FUNCTION_BLOCK FB_SlitPairV2
VAR_INPUT
    nIdPositiveAxis: UINT; //ID of axis for which positive motion increases gap size
    nIdNegativeAxis: UINT; //ID of axis for which negative motion increases gap size
    nIdGapSizeAxis: UINT; //ID of virtual gap aperture size axis
    nIdGapCentreAxis: UINT; //ID of virtual gap centre position axis

    bEnable: BOOL; //Enable slit pair logic functionality
    bReset: BOOL; //Reset from error state
    fEncoderScaling: LREAL := 10000; //Virtual axis scaling denominator, default of 10000
END_VAR
VAR
    nGapSizeEncoder AT %Q*: UDINT := 0;
    nGapCentreEncoder AT %Q*: UDINT := 0;
    fGapSize: LREAL;
    fGapCentre: LREAL;
    bAllHalted: BOOL := FALSE;
    bInternalResetHome: BOOL :=FALSE;

    fbSetpointGenEnablePositiveAxis: MC_ExtSetPointGenEnable;
    fbSetpointGenEnableNegativeAxis: MC_ExtSetPointGenEnable;
    fbSetpointGenEnableGapSizeAxis: MC_ExtSetPointGenEnable;
    fbSetpointGenEnableGapCentreAxis: MC_ExtSetPointGenEnable;

    fbSetpointGenDisablePositiveAxis: MC_ExtSetPointGenDisable;
    fbSetpointGenDisableNegativeAxis: MC_ExtSetPointGenDisable;
    fbSetpointGenDisableGapSizeAxis: MC_ExtSetPointGenDisable;
    fbSetpointGenDisableGapCentreAxis: MC_ExtSetPointGenDisable;

    fPosSetpointPositiveAxis: LREAL;
    fPosSetpointNegativeAxis: LREAL;
    fPosSetpointGapSizeAxis: LREAL;
    fPosSetpointGapCentreAxis: LREAL;
    
    fPosSetpointPositiveAxis_Last: LREAL;
    fPosSetpointNegativeAxis_Last: LREAL;
    fPosSetpointGapSizeAxis_Last: LREAL;
    fPosSetpointGapCentreAxis_Last: LREAL;
    
    fPosSetpointPositiveAxis_Nominal: LREAL;
    fPosSetpointNegativeAxis_Nominal: LREAL;
    fPosSetpointGapSizeAxis_Nominal: LREAL;
    fPosSetpointGapCentreAxis_Nominal: LREAL;
    
    fPosSetpointPositiveAxis_New: LREAL;
    fPosSetpointNegativeAxis_New: LREAL;
    fPosSetpointGapSizeAxis_New: LREAL;
    fPosSetpointGapCentreAxis_New: LREAL;

    fVeloSetpointPositiveAxis: LREAL;
    fVeloSetpointNegativeAxis: LREAL;
    fVeloSetpointGapSizeAxis: LREAL;
    fVeloSetpointGapCentreAxis: LREAL;

    fVeloSetpointPositiveAxis_New: LREAL;
    fVeloSetpointNegativeAxis_New: LREAL;
    fVeloSetpointGapSizeAxis_New: LREAL;
    fVeloSetpointGapCentreAxis_New: LREAL;
    
    nDirectionPositiveAxis: DINT;
    nDirectionNegativeAxis: DINT;
    nDirectionGapSizeAxis: DINT;
    nDirectionGapCentreAxis: DINT;
    
    ePositiveAxisState : E_AxisLimitState;
    eNegativeAxisState : E_AxisLimitState;
    eAxisPairState : E_SlitPairLimitState;
    eSlitDirectionState : E_SlitDirectionState;
    

    eState: E_SlitPairStatesV2 := E_SlitPairStatesV2.eInit;

    bInternalReset: BOOL;
    bHomingReset: BOOL := FALSE;

    //Two resets required due to homing functionality
    bResetInProgressCheck1: BOOL := FALSE;
    bResetInProgressCheck2: BOOL := FALSE;

    //internal MCPOWER blocks because Beckhoff won't let you enable a setpoint generator on a limit....
    fbPowerPositiveAxis: MC_POWER;
    fbPowerNegativeAxis: MC_POWER;
    fbPowerGapSizeAxis: MC_POWER;
    fbPowerGapCentreAxis: MC_POWER;

    //internal MC_Reset, needed because the current reset in FB_Axis works only when there is an error. This should change once the reset functionality changes
    fbInternalResetTrig: R_TRIG;
    fbInternalResetHome: R_TRIG;
    fbResetPositiveAxis: MC_RESET;
    fbResetNegativeAxis: MC_RESET;
    fbResetGapSizeAxis: MC_RESET;
    fbResetGapCentreAxis: MC_RESET;
    fbResetHomedGap: MC_Home;
    fbResetHomedCentre: MC_Home;

END_VAR

(*SETUP INSTRUCTIONS
Virtual axes:
Encoder type set to Universal
Encoder mask set to 0xFFFFFFFF
Encoder scaling set to match FB
Link nDataIn1 of encoder to FB encoders
Position lag monitoring can be left on*
Dynamics of virtual axes must be configured considering coupled mechanicals (e.g. don't set velocities your real axes can't achieve)
Virtual axis limits will need to be much more state based, for example:
GAP SIZE fwd will only be disabled if +Ve fwd hit AND -ve bwd hit, not OR
*)

//Position of virtual axes
actVirtualAxisPositions();
//Limit logic
actLimitState();
actVirtualAxisLimits();

//*NOTES*/
(*
Might need to decouple virtual axis logic (i.e. let gap size increase even if centre position locked)
Will involve untracked movements, will involve NOT enabling certain setpoint generators in certain conditions or even 
disabling and enabling other generators during moves where necessary
i.e. a limit is hit trying to full open the gap size so disabled the centre setpoint generator and "gear it in" to the real axes


*)

//Enable Logic - Virtual axes automatically enable when real axes are enabled
actVirtualAxisEnable();
//Call spGenerator FBs
actGeneratorEnableDisable();
//Calculate position setpoints
actCalculateSetpointPositions();
//Calculate velocity setpoints
//actCalculateSetpointVelocities();
//Calculate directions
actCalculateSetpointDirections();

//Error state handling - only handle errors that disable motion
IF bEnable AND (GVL.astAxes[nIdPositiveAxis].Axis.Status.ErrorStop OR GVL.astAxes[nIdNegativeAxis].Axis.Status.ErrorStop OR GVL.astAxes[nIdGapSizeAxis].Axis.Status.ErrorStop OR GVL.astAxes[nIdGapCentreAxis].Axis.Status.ErrorStop) THEN
    //eState := E_SlitPairStatesV2.eError;
END_IF

//Propagate real axis error to virtual
IF GVL.astAxes[nIdPositiveAxis].Axis.Status.ErrorStop AND (NOT GVL.astAxes[nIdGapSizeAxis].Axis.Status.ErrorStop OR NOT GVL.astAxes[nIdGapCentreAxis].Axis.Status.ErrorStop) THEN
    //GVL.astAxes[nIdGapSizeAxis].stStatus.bError := TRUE;
    //GVL.astAxes[nIdGapCentreAxis].stStatus.bError := TRUE;
    GVL.astAxes[nIdGapSizeAxis].stStatus.nErrorID := GVL.astAxes[nIdPositiveAxis].stStatus.nErrorID;
    GVL.astAxes[nIdGapCentreAxis].stStatus.nErrorID := GVL.astAxes[nIdPositiveAxis].stStatus.nErrorID;
ELSIF  GVL.astAxes[nIdNegativeAxis].Axis.Status.ErrorStop AND (NOT GVL.astAxes[nIdGapSizeAxis].Axis.Status.ErrorStop OR NOT GVL.astAxes[nIdGapCentreAxis].Axis.Status.ErrorStop) THEN
    //GVL.astAxes[nIdGapSizeAxis].stStatus.bError := TRUE;
    //GVL.astAxes[nIdGapCentreAxis].stStatus.bError := TRUE;
    GVL.astAxes[nIdGapSizeAxis].stStatus.nErrorID := GVL.astAxes[nIdNegativeAxis].stStatus.nErrorID;
    GVL.astAxes[nIdGapCentreAxis].stStatus.nErrorID := GVL.astAxes[nIdNegativeAxis].stStatus.nErrorID;
END_IF

//Internal Reset linked to any axis reset
bInternalReset := bReset OR GVL.astAxes[nIdPositiveAxis].stControl.bReset OR GVL.astAxes[nIdNegativeAxis].stControl.bReset OR GVL.astAxes[nIdGapSizeAxis].stControl.bReset OR GVL.astAxes[nIdGapCentreAxis].stControl.bReset;

//If real axis is homing, change state
IF bEnable AND (GVL.astAxes[nIdPositiveAxis].Axis.Status.HomingBusy OR GVL.astAxes[nIdNegativeAxis].Axis.Status.HomingBusy) THEN
    eState := E_SlitPairStatesV2.eWaitForRealHomed;
END_IF

//Link all halt buttons in motors
IF GVL.astAxes[nIdPositiveAxis].stControl.bHalt OR GVL.astAxes[nIdNegativeAxis].stControl.bHalt OR
    GVL.astAxes[nIdGapSizeAxis].stControl.bHalt OR GVL.astAxes[nIdGapCentreAxis].stControl.bHalt THEN
    actHaltAllAxes();
END_IF

//Propagate homing status
fbResetHomedGap(Axis:= GVL.astAxes[nIdGapSizeAxis].Axis, HomingMode:= MC_ResetCalibration);
fbResetHomedCentre(Axis:= GVL.astAxes[nIdGapCentreAxis].Axis, HomingMode:= MC_ResetCalibration);
fbInternalResetHome(CLK:= fbResetHomedCentre.Done OR fbResetHomedGap.Done );
IF NOT GVL.astAxes[nIdPositiveAxis].stStatus.bHomed OR NOT GVL.astAxes[nIdNegativeAxis].stStatus.bHomed THEN
        fbResetHomedGap.Execute := TRUE;
        fbResetHomedCentre.Execute := TRUE;
END_IF

IF fbInternalResetHome.Q THEN
        fbResetHomedGap.Execute := FALSE;
        fbResetHomedCentre.Execute := FALSE;
END_IF


//State machine
IF bEnable THEN
    CASE eState OF  //HOMING LOOP ISSUE
        E_SlitPairStatesV2.eInit:
            //If real axes are calibrated, then home the virtual axes, else go Operatioanl
            fbResetPositiveAxis(Axis:=GVL.astAxes[nIdPositiveAxis].Axis, Execute:=FALSE);
            fbResetNegativeAxis(Axis:=GVL.astAxes[nIdNegativeAxis].Axis, Execute:=FALSE);
            fbResetGapSizeAxis(Axis:=GVL.astAxes[nIdGapSizeAxis].Axis, Execute:=FALSE);
            fbResetGapCentreAxis(Axis:=GVL.astAxes[nIdGapCentreAxis].Axis, Execute:=FALSE);
            IF GVL.astAxes[nIdPositiveAxis].stStatus.bHomed AND GVL.astAxes[nIdNegativeAxis].stStatus.bHomed THEN
               GVL.astAxes[nIdGapSizeAxis].stConfig.eHomeSeq := E_HomingRoutines.eHomeDirect;
               GVL.astAxes[nIdGapCentreAxis].stConfig.eHomeSeq := E_HomingRoutines.eHomeDirect;
               GVL.astAxes[nIdGapSizeAxis].stConfig.fHomePosition := fGapSize;
               GVL.astAxes[nIdGapCentreAxis].stConfig.fHomePosition := fGapCentre;
                eState := E_SlitPairStatesV2.eWaitForVirtualHomed;
            ELSE
                eState := E_SlitPairStatesV2.eOperational;
            END_IF

        E_SlitPairStatesV2.eWaitForVirtualHomed:
            //Wait for virtual axis homing to complete/
            GVL.astAxes[nIdGapSizeAxis].stControl.eCommand := E_MotionFunctions.eHome;
            GVL.astAxes[nIdGapSizeAxis].stControl.bExecute := TRUE;
            GVL.astAxes[nIdGapCentreAxis].stControl.eCommand := E_MotionFunctions.eHome;
            GVL.astAxes[nIdGapCentreAxis].stControl.bExecute := TRUE;
            IF GVL.astAxes[nIdGapSizeAxis].stStatus.bHomed AND GVL.astAxes[nIdGapCentreAxis].stStatus.bHomed THEN
                eState := E_SlitPairStatesV2.eOperational;
            END_IF
            //IF NOT IN HOMING STATE

        E_SlitPairStatesV2.eOperational:
            bResetInProgressCheck1 := FALSE;
            //Detect whether real or virtual axes are moving
            IF GVL.astAxes[nIdGapSizeAxis].stStatus.bMoving OR GVL.astAxes[nIdGapCentreAxis].stStatus.bMoving THEN
                eState := E_SlitPairStatesV2.eEnableRealGenerators;
            END_IF
            IF GVL.astAxes[nIdPositiveAxis].stStatus.bMoving OR GVL.astAxes[nIdNegativeAxis].stStatus.bMoving THEN
                eState := E_SlitPairStatesV2.eEnableVirtualGenerators;
            END_IF

        E_SlitPairStatesV2.eEnableRealGenerators:
            //Hold MC_Power on until generators have enabled
            fbPowerPositiveAxis(Axis:=GVL.astAxes[nIdPositiveAxis].Axis, Enable:=TRUE, Enable_Positive:=TRUE,Enable_Negative:=TRUE);
            fbPowerNegativeAxis(Axis:=GVL.astAxes[nIdNegativeAxis].Axis, Enable:=TRUE, Enable_Positive:=TRUE,Enable_Negative:=TRUE);
            fbSetpointGenEnablePositiveAxis.Execute := TRUE;
            fbSetpointGenEnableNegativeAxis.Execute := TRUE;
            eState := E_SlitPairStatesV2.eCheckRealAxisGeneratorsEnabled;

        E_SlitPairStatesV2.eCheckRealAxisGeneratorsEnabled:
            //Hold MC_Power on until generators have enabled
            fbPowerPositiveAxis(Axis:=GVL.astAxes[nIdPositiveAxis].Axis, Enable:=TRUE, Enable_Positive:=TRUE,Enable_Negative:=TRUE);
            fbPowerNegativeAxis(Axis:=GVL.astAxes[nIdNegativeAxis].Axis, Enable:=TRUE, Enable_Positive:=TRUE,Enable_Negative:=TRUE);
            IF fbSetpointGenEnablePositiveAxis.Enabled AND fbSetpointGenEnableNegativeAxis.Enabled THEN
                eState := E_SlitPairStatesV2.eWaitForVirtualMoveDone;
            END_IF

        E_SlitPairStatesV2.eWaitForVirtualMoveDone:            
            IF NOT(GVL.astAxes[nIdGapSizeAxis].stStatus.bMoving OR GVL.astAxes[nIdGapCentreAxis].stStatus.bMoving) THEN
                eState := E_SlitPairStatesV2.eDisableRealGenerators;
            END_IF

        E_SlitPairStatesV2.eDisableRealGenerators:
            fbSetpointGenDisablePositiveAxis.Execute := TRUE;
            fbSetpointGenDisableNegativeAxis.Execute := TRUE;
            eState := E_SlitPairStatesV2.eOperational;

        E_SlitPairStatesV2.eEnableVirtualGenerators:
            //Hold MC_Power on until generators have enabled
            fbPowerGapSizeAxis(Axis:=GVL.astAxes[nIdGapSizeAxis].Axis, Enable:=TRUE, Enable_Positive:=TRUE,Enable_Negative:=TRUE);
            fbPowerGapCentreAxis(Axis:=GVL.astAxes[nIdGapCentreAxis].Axis, Enable:=TRUE, Enable_Positive:=TRUE,Enable_Negative:=TRUE);
            fbSetpointGenEnableGapSizeAxis.Execute := TRUE;
            fbSetpointGenEnableGapCentreAxis.Execute := TRUE;
            eState := E_SlitPairStatesV2.eCheckVirtualAxisGeneratorsEnabled;

        E_SlitPairStatesV2.eCheckVirtualAxisGeneratorsEnabled:
            //Hold MC_Power on until generators have enabled
            fbPowerGapSizeAxis(Axis:=GVL.astAxes[nIdGapSizeAxis].Axis, Enable:=TRUE, Enable_Positive:=TRUE,Enable_Negative:=TRUE);
            fbPowerGapCentreAxis(Axis:=GVL.astAxes[nIdGapCentreAxis].Axis, Enable:=TRUE, Enable_Positive:=TRUE,Enable_Negative:=TRUE);
            IF fbSetpointGenEnableGapSizeAxis.Enabled AND fbSetpointGenEnableGapCentreAxis.Enabled THEN
                eState := E_SlitPairStatesV2.eWaitForRealMoveDone;
            END_IF

        E_SlitPairStatesV2.eWaitForRealMoveDone:
            IF NOT(GVL.astAxes[nIdPositiveAxis].stStatus.bMoving OR GVL.astAxes[nIdNegativeAxis].stStatus.bMoving) THEN
                eState := E_SlitPairStatesV2.eDisableVirtualGenerators;
            END_IF

        E_SlitPairStatesV2.eDisableVirtualGenerators:
            fbSetpointGenDisableGapSizeAxis.Execute := TRUE;
            fbSetpointGenDisableGapCentreAxis.Execute := TRUE;
            eState := E_SlitPairStatesV2.eOperational;

        E_SlitPairStatesV2.eError:
            actHaltAllAxes();

            IF bHomingReset THEN
                bInternalReset := TRUE;
                bResetInProgressCheck1 := TRUE;
                bResetInProgressCheck2 := TRUE;
                bHomingReset := FALSE;
            END_IF
            IF bInternalReset OR bReset OR bResetInProgressCheck2 THEN
                fbResetPositiveAxis(Axis:=GVL.astAxes[nIdPositiveAxis].Axis, Execute:=TRUE);
                fbResetNegativeAxis(Axis:=GVL.astAxes[nIdNegativeAxis].Axis, Execute:=TRUE);
                fbResetGapSizeAxis(Axis:=GVL.astAxes[nIdGapSizeAxis].Axis, Execute:=TRUE);
                fbResetGapCentreAxis(Axis:=GVL.astAxes[nIdGapCentreAxis].Axis, Execute:=TRUE);
                GVL.astAxes[nIdPositiveAxis].stControl.bReset := TRUE;
                GVL.astAxes[nIdNegativeAxis].stControl.bReset := TRUE;
                GVL.astAxes[nIdGapSizeAxis].stControl.bReset := TRUE;
                GVL.astAxes[nIdGapCentreAxis].stControl.bReset := TRUE;
                IF NOT(bResetInProgressCheck1) THEN
                    bResetInProgressCheck2 := FALSE;
                END_IF
            END_IF

            IF NOT(GVL.astAxes[nIdPositiveAxis].stStatus.bError) AND NOT(GVL.astAxes[nIdNegativeAxis].stStatus.bError) AND NOT(GVL.astAxes[nIdGapSizeAxis].stStatus.bError) AND NOT(GVL.astAxes[nIdGapCentreAxis].stStatus.bError) THEN
                eState := E_SlitPairStatesV2.eInit;
            END_IF

        E_SlitPairStatesV2.eWaitForRealHomed:
            bHomingReset := TRUE;
            IF NOT GVL.astAxes[nIdPositiveAxis].Axis.Status.Homed OR NOT GVL.astAxes[nIdNegativeAxis].Axis.Status.Homed THEN
                eState := E_SlitPairStatesV2.eInit;
            END_IF
    END_CASE
END_IF


//Feed externalsetpoint generators setpoint values - ignoring acceleration
MC_ExtSetPointGenFeed(Axis:= GVL.astAxes[nIdPositiveAxis].Axis, Position:= fPosSetpointPositiveAxis, Velocity:= fVeloSetpointPositiveAxis, Acceleration:= 0, Direction:= nDirectionPositiveAxis);
MC_ExtSetPointGenFeed(Axis:= GVL.astAxes[nIdNegativeAxis].Axis, Position:= fPosSetpointNegativeAxis, Velocity:= fVeloSetpointNegativeAxis, Acceleration:= 0, Direction:= nDirectionNegativeAxis);
MC_ExtSetPointGenFeed(Axis:= GVL.astAxes[nIdGapSizeAxis].Axis, Position:= fPosSetpointGapSizeAxis, Velocity:= fVeloSetpointGapSizeAxis, Acceleration:= 0, Direction:= nDirectionGapSizeAxis);
MC_ExtSetPointGenFeed(Axis:= GVL.astAxes[nIdGapCentreAxis].Axis, Position:= fPosSetpointGapCentreAxis, Velocity:= fVeloSetpointGapCentreAxis, Acceleration:= 0, Direction:= nDirectionGapCentreAxis);

bReset := FALSE;

ACTION actCalculateSetpointDirections:

IF fVeloSetpointPositiveAxis > 0 THEN
    nDirectionPositiveAxis := 1; //moving forward
ELSIF fVeloSetpointPositiveAxis < 0 THEN
    nDirectionPositiveAxis := -1; //moving backward
ELSE
    nDirectionPositiveAxis := 0; //stationary
END_IF

IF fVeloSetpointNegativeAxis > 0 THEN
    nDirectionNegativeAxis := 1; //moving forward
ELSIF fVeloSetpointNegativeAxis < 0 THEN
    nDirectionNegativeAxis := -1; //moving backward
ELSE
    nDirectionNegativeAxis := 0; //stationary
END_IF

IF fVeloSetpointGapSizeAxis > 0 THEN
    nDirectionGapSizeAxis := 1; //moving forward
ELSIF fVeloSetpointGapSizeAxis < 0 THEN
    nDirectionGapSizeAxis := -1; //moving backward
ELSE
    nDirectionGapSizeAxis := 0; //stationary
END_IF

IF fVeloSetpointGapCentreAxis > 0 THEN
    nDirectionGapCentreAxis := 1; //moving forward
ELSIF fVeloSetpointGapCentreAxis < 0 THEN
    nDirectionGapCentreAxis := -1; //moving backward
ELSE
    nDirectionGapCentreAxis := 0; //stationary
END_IF
END_ACTION

ACTION actCalculateSetpointPositions:
GVL.astAxes[nIdPositiveAxis].Axis.ReadStatus();
GVL.astAxes[nIdNegativeAxis].Axis.ReadStatus();
GVL.astAxes[nIdGapSizeAxis].Axis.ReadStatus();
GVL.astAxes[nIdGapCentreAxis].Axis.ReadStatus();





//Generate the NEW setpoint positions as if everything was hunky-dory
fPosSetpointPositiveAxis_Nominal := GVL.astAxes[nIdGapCentreAxis].Axis.NcToPlc.SetPos + (GVL.astAxes[nIdGapSizeAxis].Axis.NcToPlc.SetPos/2);
fPosSetpointNegativeAxis_Nominal := GVL.astAxes[nIdGapCentreAxis].Axis.NcToPlc.SetPos - (GVL.astAxes[nIdGapSizeAxis].Axis.NcToPlc.SetPos/2);
fPosSetpointGapSizeAxis_Nominal := GVL.astAxes[nIdPositiveAxis].Axis.NcToPlc.SetPos - GVL.astAxes[nIdNegativeAxis].Axis.NcToPlc.SetPos;
fPosSetpointGapCentreAxis_Nominal := (GVL.astAxes[nIdPositiveAxis].Axis.NcToPlc.SetPos + GVL.astAxes[nIdNegativeAxis].Axis.NcToPlc.SetPos) / 2;


//Update previous nominal
//fPosSetpointPositiveAxis_Nominal:= fPosSetpointPositiveAxis_New;
//fPosSetpointNegativeAxis_Nominal:= fPosSetpointNegativeAxis_New;
//fPosSetpointGapSizeAxis_Nominal:= fPosSetpointGapSizeAxis_New;
//fPosSetpointGapCentreAxis_Nominal:= fPosSetpointGapCentreAxis_New;



(*//Set direction state of slit
IF fPosSetpointPositiveAxis_New>fPosSetpointPositiveAxis_Nominal THEN
    //PositiveFwd
    IF fPosSetpointNegativeAxis_New>fPosSetpointNegativeAxis_Nominal THEN
        eSlitDirectionState:= E_SlitDirectionState.PositiveFwd_NegativeFwd;
    ELSIF fPosSetpointNegativeAxis_New < fPosSetpointNegativeAxis_Nominal THEN
        eSlitDirectionState:= E_SlitDirectionState.PositiveFwd_NegativeBwd;
    ELSE
        eSlitDirectionState:= E_SlitDirectionState.PositiveFwd_NegativeStationary;
	END_IF
ELSIF fPosSetpointPositiveAxis_New<fPosSetpointPositiveAxis_Nominal THEN    
    //PositiveBwd
    IF fPosSetpointNegativeAxis_New>fPosSetpointNegativeAxis_Nominal THEN
        eSlitDirectionState:= E_SlitDirectionState.PositiveBwd_NegativeFwd;
    ELSIF fPosSetpointNegativeAxis_New < fPosSetpointNegativeAxis_Nominal THEN
        eSlitDirectionState:= E_SlitDirectionState.PositiveBwd_NegativeBwd;
    ELSE
        eSlitDirectionState:= E_SlitDirectionState.PositiveBwd_NegativeStationary;
	END_IF
ELSE
    //PositiveStationary
    IF fPosSetpointNegativeAxis_New>fPosSetpointNegativeAxis_Nominal THEN
        eSlitDirectionState:= E_SlitDirectionState.PositiveStationary_NegativeFwd;
    ELSIF fPosSetpointNegativeAxis_New < fPosSetpointNegativeAxis_Nominal THEN
        eSlitDirectionState:= E_SlitDirectionState.PositiveStationary_NegativeBwd;
    ELSE
        eSlitDirectionState:= E_SlitDirectionState.PositiveStationary_NegativeStationary;
	END_IF
END_IF*)







fVeloSetpointPositiveAxis_New := GVL.astAxes[nIdGapCentreAxis].Axis.NcToPlc.SetVelo +(GVL.astAxes[nIdGapSizeAxis].Axis.NcToPlc.SetVelo/2);
IF ABS(fVeloSetpointPositiveAxis_New) < 0.01 THEN
    fVeloSetpointPositiveAxis_New:=0;
END_IF
fVeloSetpointNegativeAxis_New := GVL.astAxes[nIdGapCentreAxis].Axis.NcToPlc.SetVelo -(GVL.astAxes[nIdGapSizeAxis].Axis.NcToPlc.SetVelo/2);
IF ABS(fVeloSetpointNegativeAxis_New) < 0.01 THEN
    fVeloSetpointNegativeAxis_New:=0;
END_IF
fVeloSetpointGapSizeAxis_New := GVL.astAxes[nIdPositiveAxis].Axis.NcToPlc.SetVelo - GVL.astAxes[nIdNegativeAxis].Axis.NcToPlc.SetVelo;
IF ABS(fVeloSetpointGapSizeAxis_New) < 0.01 THEN
    fVeloSetpointGapSizeAxis_New:=0;
END_IF
fVeloSetpointGapCentreAxis_New := GVL.astAxes[nIdPositiveAxis].Axis.NcToPlc.SetVelo + GVL.astAxes[nIdNegativeAxis].Axis.NcToPlc.SetVelo;
IF ABS(fVeloSetpointGapCentreAxis_New) < 0.01 THEN
    fVeloSetpointGapCentreAxis_New:=0;
END_IF

//IF THE REAL AXES ARE BEING CONTROLLED BY AN EXTERNAL SETPOINT GENERATOR i.e. THE VIRTUAL AXES IN CONTROL
IF GVL.astAxes[nIdPositiveAxis].Axis.Status.ExtSetPointGenEnabled OR GVL.astAxes[nIdNegativeAxis].Axis.Status.ExtSetPointGenEnabled THEN
    IF GVL.astAxes[nIdGapSizeAxis].Axis.Status.PositiveDirection THEN
        CASE eAxisPairState OF            
        E_SlitPairLimitState.PositiveOnForward_NegativeOnForward:
            Setpoint_PositiveDisabled();

        E_SlitPairLimitState.PositiveOnForward_NegativeOnBackward:
            Setpoint_AllDisabled();
            
        E_SlitPairLimitState.PositiveOnForward_NegativeOnNoLimit:
            Setpoint_PositiveDisabled();
            
        E_SlitPairLimitState.PositiveOnBackward_NegativeOnForward:
            Setpoint_Normal();
            
        E_SlitPairLimitState.PositiveOnBackward_NegativeOnBackward:
            Setpoint_NegativeDisabled();
            
        E_SlitPairLimitState.PositiveOnBackward_NegativeOnNoLimit:
            Setpoint_Normal();
            
        E_SlitPairLimitState.PositiveOnNoLimit_NegativeOnForward:
            Setpoint_Normal();
            
        E_SlitPairLimitState.PositiveOnNoLimit_NegativeOnBackward:
            Setpoint_NegativeDisabled();
            
        E_SlitPairLimitState.PositiveOnNoLimit_NegativeOnNoLimit:
            Setpoint_Normal();                       
        END_CASE
    ELSIF GVL.astAxes[nIdGapSizeAxis].Axis.Status.NegativeDirection THEN
        CASE eAxisPairState OF            
        E_SlitPairLimitState.PositiveOnForward_NegativeOnForward:
            Setpoint_NegativeDisabled();

        E_SlitPairLimitState.PositiveOnForward_NegativeOnBackward:
            Setpoint_Normal();
            
        E_SlitPairLimitState.PositiveOnForward_NegativeOnNoLimit:
            Setpoint_Normal();
            
        E_SlitPairLimitState.PositiveOnBackward_NegativeOnForward:
            Setpoint_AllDisabled();
            
        E_SlitPairLimitState.PositiveOnBackward_NegativeOnBackward:
            Setpoint_PositiveDisabled();
            
        E_SlitPairLimitState.PositiveOnBackward_NegativeOnNoLimit:
            Setpoint_PositiveDisabled();
            
        E_SlitPairLimitState.PositiveOnNoLimit_NegativeOnForward:
            Setpoint_NegativeDisabled();
            
        E_SlitPairLimitState.PositiveOnNoLimit_NegativeOnBackward:
            Setpoint_Normal();
            
        E_SlitPairLimitState.PositiveOnNoLimit_NegativeOnNoLimit:
            Setpoint_Normal();                       
        END_CASE
    ELSE
        //GAP CENTRE MOVING
        IF GVL.astAxes[nIdGapCentreAxis].Axis.Status.PositiveDirection THEN
            CASE eAxisPairState OF            
            E_SlitPairLimitState.PositiveOnForward_NegativeOnForward:
                Setpoint_AllDisabled();

            E_SlitPairLimitState.PositiveOnForward_NegativeOnBackward:
                Setpoint_AllDisabled();
            
            E_SlitPairLimitState.PositiveOnForward_NegativeOnNoLimit:
                Setpoint_AllDisabled();
            
            E_SlitPairLimitState.PositiveOnBackward_NegativeOnForward:
                Setpoint_AllDisabled();
            
            E_SlitPairLimitState.PositiveOnBackward_NegativeOnBackward:
                Setpoint_Normal();
            
            E_SlitPairLimitState.PositiveOnBackward_NegativeOnNoLimit:
                Setpoint_Normal();
            
            E_SlitPairLimitState.PositiveOnNoLimit_NegativeOnForward:
                Setpoint_AllDisabled();
            
            E_SlitPairLimitState.PositiveOnNoLimit_NegativeOnBackward:
                Setpoint_Normal();
            
            E_SlitPairLimitState.PositiveOnNoLimit_NegativeOnNoLimit:
                Setpoint_Normal();                       
            END_CASE
        ELSIF GVL.astAxes[nIdGapCentreAxis].Axis.Status.NegativeDirection THEN
            CASE eAxisPairState OF            
            E_SlitPairLimitState.PositiveOnForward_NegativeOnForward:
                Setpoint_Normal();

            E_SlitPairLimitState.PositiveOnForward_NegativeOnBackward:
                Setpoint_AllDisabled();
            
            E_SlitPairLimitState.PositiveOnForward_NegativeOnNoLimit:
                Setpoint_Normal();
            
            E_SlitPairLimitState.PositiveOnBackward_NegativeOnForward:
                Setpoint_AllDisabled();
            
            E_SlitPairLimitState.PositiveOnBackward_NegativeOnBackward:
                Setpoint_AllDisabled();
            
            E_SlitPairLimitState.PositiveOnBackward_NegativeOnNoLimit:
                Setpoint_AllDisabled();
            
            E_SlitPairLimitState.PositiveOnNoLimit_NegativeOnForward:
                Setpoint_Normal();
            
            E_SlitPairLimitState.PositiveOnNoLimit_NegativeOnBackward:
                Setpoint_AllDisabled();
            
            E_SlitPairLimitState.PositiveOnNoLimit_NegativeOnNoLimit:
                Setpoint_Normal();                       
            END_CASE
		END_IF
    END_IF
ELSE
    //OTHER DIRECTIONS HERE
   // fVeloSetpointPositiveAxis := fVeloSetpointPositiveAxis_New;
    //fVeloSetpointNegativeAxis := fVeloSetpointNegativeAxis_New;
    fVeloSetpointGapSizeAxis := fVeloSetpointGapSizeAxis_New;
    fVeloSetpointGapCentreAxis := fVeloSetpointGapCentreAxis_New;
END_IF

    



IF GVL.astAxes[nIdGapCentreAxis].Axis.Status.ExtSetPointGenEnabled AND GVL.astAxes[nIdGapSizeAxis].Axis.Status.ExtSetPointGenEnabled THEN
    fPosSetpointGapSizeAxis := GVL.astAxes[nIdPositiveAxis].Axis.NcToPlc.SetPos - GVL.astAxes[nIdNegativeAxis].Axis.NcToPlc.SetPos;
    fPosSetpointGapCentreAxis := (GVL.astAxes[nIdPositiveAxis].Axis.NcToPlc.SetPos + GVL.astAxes[nIdNegativeAxis].Axis.NcToPlc.SetPos) / 2;
    fVeloSetpointGapCentreAxis := fVeloSetpointGapCentreAxis_New;
    fVeloSetpointGapSizeAxis := fVeloSetpointGapSizeAxis_New;
END_IF





//Nominal last positions for determining direction
fPosSetpointPositiveAxis_Last := fPosSetpointPositiveAxis_Nominal; //GVL.astAxes[nIdPositiveAxis].Axis.NcToPlc.SetPos;
fPosSetpointNegativeAxis_Last := fPosSetpointNegativeAxis_Nominal;//GVL.astAxes[nIdNegativeAxis].Axis.NcToPlc.SetPos;
fPosSetpointGapSizeAxis_Last := fPosSetpointGapSizeAxis_Nominal; //GVL.astAxes[nIdGapSizeAxis].Axis.NcToPlc.SetPos;
fPosSetpointGapCentreAxis_Last := fPosSetpointGapCentreAxis_Nominal; //GVL.astAxes[nIdGapCentreAxis].Axis.NcToPlc.SetPos;








(*BACKUP
IF GVL.astAxes[nIdPositiveAxis].Axis.Status.ExtSetPointGenEnabled AND GVL.astAxes[nIdNegativeAxis].Axis.Status.ExtSetPointGenEnabled THEN
    IF fPosSetpointPositiveAxis_New > GVL.astAxes[nIdPositiveAxis].Axis.NcToPlc.ActPos AND GVL.astAxes[nIdPositiveAxis].stInputs.bLimitFwd = FALSE THEN
    fPosSetpointPositiveAxis := fPosSetpointPositiveAxis;
    fbSetpointGenEnableGapCentreAxis.Execute:= TRUE;
    ELSE
        fPosSetpointPositiveAxis := GVL.astAxes[nIdGapCentreAxis].Axis.NcToPlc.SetPos + (GVL.astAxes[nIdGapSizeAxis].Axis.NcToPlc.SetPos/2);
    END_IF



    IF fPosSetpointNegativeAxis_New < GVL.astAxes[nIdNegativeAxis].Axis.NcToPlc.ActPos AND GVL.astAxes[nIdNegativeAxis].stInputs.bLimitBwd = FALSE THEN
        fPosSetpointNegativeAxis := fPosSetpointNegativeAxis;
        fbSetpointGenEnableGapCentreAxis.Execute:= TRUE;
    ELSE
        fPosSetpointNegativeAxis := GVL.astAxes[nIdGapCentreAxis].Axis.NcToPlc.SetPos - (GVL.astAxes[nIdGapSizeAxis].Axis.NcToPlc.SetPos/2);
    END_IF

END_IF
*)

(* //ORIGINAL CODE
fPosSetpointPositiveAxis := GVL.astAxes[nIdGapCentreAxis].Axis.NcToPlc.SetPos + (GVL.astAxes[nIdGapSizeAxis].Axis.NcToPlc.SetPos/2);
fPosSetpointNegativeAxis := GVL.astAxes[nIdGapCentreAxis].Axis.NcToPlc.SetPos - (GVL.astAxes[nIdGapSizeAxis].Axis.NcToPlc.SetPos/2);

fPosSetpointGapSizeAxis := GVL.astAxes[nIdPositiveAxis].Axis.NcToPlc.SetPos - GVL.astAxes[nIdNegativeAxis].Axis.NcToPlc.SetPos;
fPosSetpointGapCentreAxis := (GVL.astAxes[nIdPositiveAxis].Axis.NcToPlc.SetPos + GVL.astAxes[nIdNegativeAxis].Axis.NcToPlc.SetPos) / 2;

*)
END_ACTION

ACTION actCalculateSetpointVelocities:
(*IF fPosSetpointGapSizeAxis_Last > fPosSetpointGapSizeAxis THEN
    //If NEGATIVE axis on BWD limit AND POSTIVE Axis NOT on FWD LIMIT - LET POSITIVE AXIS MOVE
    IF GVL.astAxes[nIdNegativeAxis].stStatus.bBwEnabled = FALSE AND GVL.astAxes[nIdPositiveAxis].stStatus.bFwEnabled THEN
        fVeloSetpointPositiveAxis := GVL.astAxes[nIdGapCentreAxis].Axis.NcToPlc.SetVelo +(GVL.astAxes[nIdGapSizeAxis].Axis.NcToPlc.SetVelo);
        fVeloSetpointNegativeAxis := 0;
        
   //If POSTIVE axis on FWD limit AND NEGATIVE Axis NOT on BWD LIMIT - LET NEGATIVE AXIS MOVE
    ELSIF GVL.astAxes[nIdPositiveAxis].stStatus.bFwEnabled = FALSE AND GVL.astAxes[nIdNegativeAxis].stStatus.bBwEnabled THEN
        fVeloSetpointPositiveAxis := 0;
        fVeloSetpointNegativeAxis := GVL.astAxes[nIdGapCentreAxis].Axis.NcToPlc.SetVelo -(GVL.astAxes[nIdGapSizeAxis].Axis.NcToPlc.SetVelo/2);
        
    //If POSTIVE axis NOT on FWD limit AND NEGATIVE Axis NOT on BWD LIMIT - NORMAL OPERATION
    ELSIF GVL.astAxes[nIdPositiveAxis].stStatus.bFwEnabled AND GVL.astAxes[nIdNegativeAxis].stStatus.bBwEnabled THEN
        fVeloSetpointPositiveAxis := GVL.astAxes[nIdGapCentreAxis].Axis.NcToPlc.SetVelo +(GVL.astAxes[nIdGapSizeAxis].Axis.NcToPlc.SetVelo/2);
        fVeloSetpointNegativeAxis := GVL.astAxes[nIdGapCentreAxis].Axis.NcToPlc.SetVelo -(GVL.astAxes[nIdGapSizeAxis].Axis.NcToPlc.SetVelo/2);
        
    //If POSTIVE axis on FWD limit AND NEGATIVE Axis  on BWD LIMIT  - DON'T MOVE
    ELSIF GVL.astAxes[nIdNegativeAxis].stStatus.bBwEnabled = FALSE AND GVL.astAxes[nIdPositiveAxis].stStatus.bFwEnabled = FALSE THEN
        fVeloSetpointPositiveAxis := 0;
        fPosSetpointNegativeAxis := 0;
	END_IF
END_IF

//GAP SIZE GETTING SMALLER
IF fPosSetpointGapSizeAxis_Last < fPosSetpointGapSizeAxis THEN
    //If NEGATIVE axis on FWD limit AND POSTIVE Axis NOT on BWD LIMIT - LET POSITIVE AXIS MOVE
    IF GVL.astAxes[nIdNegativeAxis].stStatus.bFwEnabled = FALSE AND GVL.astAxes[nIdPositiveAxis].stStatus.bBwEnabled THEN
        fVeloSetpointPositiveAxis := GVL.astAxes[nIdGapCentreAxis].Axis.NcToPlc.SetVelo +(GVL.astAxes[nIdGapSizeAxis].Axis.NcToPlc.SetVelo);
        fVeloSetpointNegativeAxis := 0;
        
   //If POSTIVE axis on BWD limit AND NEGATIVE Axis NOT on FWD LIMIT - LET NEGATIVE AXIS MOVE
    ELSIF GVL.astAxes[nIdPositiveAxis].stStatus.bBwEnabled = FALSE AND GVL.astAxes[nIdNegativeAxis].stStatus.bFwEnabled THEN
        fVeloSetpointPositiveAxis := 0;
        fVeloSetpointNegativeAxis := GVL.astAxes[nIdGapCentreAxis].Axis.NcToPlc.SetVelo -(GVL.astAxes[nIdGapSizeAxis].Axis.NcToPlc.SetVelo/2);
 
    //If POSTIVE axis NOT on BWD limit AND NEGATIVE Axis NOT on FWD LIMIT - NORMAL OPERATION
    ELSIF GVL.astAxes[nIdPositiveAxis].stStatus.bBwEnabled AND GVL.astAxes[nIdNegativeAxis].stStatus.bFwEnabled THEN
        fVeloSetpointPositiveAxis := GVL.astAxes[nIdGapCentreAxis].Axis.NcToPlc.SetVelo +(GVL.astAxes[nIdGapSizeAxis].Axis.NcToPlc.SetVelo/2);
        fVeloSetpointNegativeAxis := GVL.astAxes[nIdGapCentreAxis].Axis.NcToPlc.SetVelo -(GVL.astAxes[nIdGapSizeAxis].Axis.NcToPlc.SetVelo/2);
        
    //If POSTIVE axis on BWD limit AND NEGATIVE Axis  on FWD LIMIT  - DON'T MOVE
    ELSIF GVL.astAxes[nIdNegativeAxis].stStatus.bFwEnabled = FALSE AND GVL.astAxes[nIdPositiveAxis].stStatus.bBwEnabled = FALSE THEN
        fVeloSetpointPositiveAxis := 0;
        fPosSetpointNegativeAxis := 0;
	END_IF
END_IF*)




fVeloSetpointPositiveAxis := GVL.astAxes[nIdGapCentreAxis].Axis.NcToPlc.SetVelo +(GVL.astAxes[nIdGapSizeAxis].Axis.NcToPlc.SetVelo/2);
fVeloSetpointNegativeAxis := GVL.astAxes[nIdGapCentreAxis].Axis.NcToPlc.SetVelo -(GVL.astAxes[nIdGapSizeAxis].Axis.NcToPlc.SetVelo/2);
fVeloSetpointGapSizeAxis := GVL.astAxes[nIdPositiveAxis].Axis.NcToPlc.SetVelo - GVL.astAxes[nIdNegativeAxis].Axis.NcToPlc.SetVelo;
fVeloSetpointGapCentreAxis := GVL.astAxes[nIdPositiveAxis].Axis.NcToPlc.SetVelo + GVL.astAxes[nIdNegativeAxis].Axis.NcToPlc.SetVelo;


IF ABS(fPosSetpointPositiveAxis_Last-fPosSetpointPositiveAxis)<0.001 THEN
    fVeloSetpointPositiveAxis := 0;
END_IF

IF ABS(fPosSetpointNegativeAxis_Last-fPosSetpointNegativeAxis)<0.001 THEN
    fVeloSetpointNegativeAxis := 0;
END_IF
END_ACTION

ACTION actGeneratorEnableDisable:

fbSetpointGenEnablePositiveAxis(Axis:=GVL.astAxes[nIdPositiveAxis].Axis);
fbSetpointGenEnablePositiveAxis.Execute := FALSE;

fbSetpointGenEnableNegativeAxis(Axis:=GVL.astAxes[nIdNegativeAxis].Axis);
fbSetpointGenEnableNegativeAxis.Execute := FALSE;

fbSetpointGenEnableGapSizeAxis(Axis:=GVL.astAxes[nIdGapSizeAxis].Axis);
fbSetpointGenEnableGapSizeAxis.Execute := FALSE;

fbSetpointGenEnableGapCentreAxis(Axis:=GVL.astAxes[nIdGapCentreAxis].Axis);
fbSetpointGenEnableGapCentreAxis.Execute := FALSE;


fbSetpointGenDisablePositiveAxis(Axis:=GVL.astAxes[nIdPositiveAxis].Axis);
fbSetpointGenDisablePositiveAxis.Execute := FALSE;

fbSetpointGenDisableNegativeAxis(Axis:=GVL.astAxes[nIdNegativeAxis].Axis);
fbSetpointGenDisableNegativeAxis.Execute := FALSE;

fbSetpointGenDisableGapSizeAxis(Axis:=GVL.astAxes[nIdGapSizeAxis].Axis);
fbSetpointGenDisableGapSizeAxis.Execute := FALSE;

fbSetpointGenDisableGapCentreAxis(Axis:=GVL.astAxes[nIdGapCentreAxis].Axis);
fbSetpointGenDisableGapCentreAxis.Execute := FALSE;
END_ACTION

ACTION actHaltAllAxes:

GVL.astAxes[nIdPositiveAxis].stControl.bHalt := TRUE;
GVL.astAxes[nIdNegativeAxis].stControl.bHalt := TRUE;
GVL.astAxes[nIdGapSizeAxis].stControl.bHalt := TRUE;
GVL.astAxes[nIdGapCentreAxis].stControl.bHalt := TRUE;
bAllHalted := TRUE;

//Reset Halts
IF bAllHalted AND NOT GVL.astAxes[nIdPositiveAxis].stStatus.bMoving AND NOT GVL.astAxes[nIdNegativeAxis].stStatus.bMoving
 AND NOT GVL.astAxes[nIdGapSizeAxis].stStatus.bMoving AND NOT GVL.astAxes[nIdGapCentreAxis].stStatus.bMoving THEN
   GVL.astAxes[nIdPositiveAxis].stControl.bHalt := FALSE;
   GVL.astAxes[nIdNegativeAxis].stControl.bHalt := FALSE;
   GVL.astAxes[nIdGapSizeAxis].stControl.bHalt := FALSE;
   GVL.astAxes[nIdGapCentreAxis].stControl.bHalt := FALSE;
   bAllHalted := FALSE;
END_IF
END_ACTION

ACTION actLimitState:
//Positive axis state
IF GVL.astAxes[nIdPositiveAxis].stInputs.bLimitFwd = FALSE THEN
    ePositiveAxisState := E_AxisLimitState.OnForwardLimit;
ELSIF GVL.astAxes[nIdPositiveAxis].stInputs.bLimitBwd = FALSE THEN
    ePositiveAxisState := E_AxisLimitState.OnBackwardLimit;
ELSE
    ePositiveAxisState := E_AxisLimitState.NoLimit;
END_IF

//Negative axis state
IF GVL.astAxes[nIdNegativeAxis].stInputs.bLimitFwd = FALSE THEN
    eNegativeAxisState := E_AxisLimitState.OnForwardLimit;
ELSIF GVL.astAxes[nIdNegativeAxis].stInputs.bLimitBwd = FALSE THEN
    eNegativeAxisState := E_AxisLimitState.OnBackwardLimit;
ELSE
    eNegativeAxisState := E_AxisLimitState.NoLimit;
END_IF



CASE ePositiveAxisState OF
    E_AxisLimitState.OnForwardLimit:
        CASE eNegativeAxisState OF
            E_AxisLimitState.OnForwardLimit:
                eAxisPairState := E_SlitPairLimitState.PositiveOnForward_NegativeOnForward;
            E_AxisLimitState.OnBackwardLimit:
                eAxisPairState := E_SlitPairLimitState.PositiveOnForward_NegativeOnBackward;
            E_AxisLimitState.NoLimit:
                eAxisPairState := E_SlitPairLimitState.PositiveOnForward_NegativeOnNoLimit;            
		END_CASE
    E_AxisLimitState.OnBackwardLimit:
        CASE eNegativeAxisState OF
            E_AxisLimitState.OnForwardLimit:
                eAxisPairState := E_SlitPairLimitState.PositiveOnBackward_NegativeOnForward;
            E_AxisLimitState.OnBackwardLimit:
                eAxisPairState := E_SlitPairLimitState.PositiveOnBackward_NegativeOnBackward;
            E_AxisLimitState.NoLimit:
                eAxisPairState := E_SlitPairLimitState.PositiveOnBackward_NegativeOnNoLimit;            
		END_CASE
    E_AxisLimitState.NoLimit:
        CASE eNegativeAxisState OF
            E_AxisLimitState.OnForwardLimit:
                eAxisPairState := E_SlitPairLimitState.PositiveOnNoLimit_NegativeOnForward;
            E_AxisLimitState.OnBackwardLimit:
                eAxisPairState := E_SlitPairLimitState.PositiveOnNoLimit_NegativeOnBackward;
            E_AxisLimitState.NoLimit:
                eAxisPairState := E_SlitPairLimitState.PositiveOnNoLimit_NegativeOnNoLimit;            
		END_CASE
END_CASE
END_ACTION

ACTION actVirtualAxisEnable:
GVL.astAxes[nIdGapSizeAxis].stControl.bEnable := GVL.astAxes[nIdPositiveAxis].stControl.bEnable AND GVL.astAxes[nIdNegativeAxis].stControl.bEnable;
GVL.astAxes[nIdGapCentreAxis].stControl.bEnable := GVL.astAxes[nIdPositiveAxis].stControl.bEnable AND GVL.astAxes[nIdNegativeAxis].stControl.bEnable;

//GVL.astAxes[nIdGapSizeAxis].stControl.bEnable := GVL.astAxes[nIdPositiveAxis].stStatus.bEnabled AND GVL.astAxes[nIdNegativeAxis].stStatus.bEnabled;
//GVL.astAxes[nIdGapCentreAxis].stControl.bEnable := GVL.astAxes[nIdPositiveAxis].stStatus.bEnabled AND GVL.astAxes[nIdNegativeAxis].stStatus.bEnabled;
END_ACTION

ACTION actVirtualAxisLimits:
//GAP SIZE FORWARD LIMIT
IF GVL.astAxes[nIdPositiveAxis].stStatus.bFwEnabled = FALSE AND GVL.astAxes[nIdNegativeAxis].stStatus.bBwEnabled = FALSE THEN
    //GVL.astAxes[nIdGapSizeAxis].stInputs.bLimitFwd := FALSE;
    GVL.astAxes[nIdGapSizeAxis].stStatus.bFwEnabled := FALSE;
ELSE
    //GVL.astAxes[nIdGapSizeAxis].stInputs.bLimitFwd := TRUE;
    GVL.astAxes[nIdGapSizeAxis].stStatus.bFwEnabled := TRUE;
END_IF

//GAP SIZE BACKWARD LIMIT
IF GVL.astAxes[nIdPositiveAxis].stStatus.bBwEnabled = FALSE AND GVL.astAxes[nIdNegativeAxis].stStatus.bFwEnabled = FALSE THEN
    //GVL.astAxes[nIdGapSizeAxis].stInputs.bLimitBwd := FALSE;
    GVL.astAxes[nIdGapSizeAxis].stStatus.bBwEnabled := FALSE;
ELSE
    //GVL.astAxes[nIdGapSizeAxis].stInputs.bLimitBwd := TRUE;
    GVL.astAxes[nIdGapSizeAxis].stStatus.bBwEnabled := TRUE;
END_IF

//GAP CENTRE FORWARD LIMIT
IF GVL.astAxes[nIdPositiveAxis].stStatus.bFwEnabled = FALSE OR GVL.astAxes[nIdNegativeAxis].stStatus.bFwEnabled = FALSE THEN
    //GVL.astAxes[nIdGapCentreAxis].stInputs.bLimitFwd := FALSE;
    GVL.astAxes[nIdGapCentreAxis].stStatus.bFwEnabled := FALSE;
ELSE
    //GVL.astAxes[nIdGapCentreAxis].stInputs.bLimitFwd := TRUE;
    GVL.astAxes[nIdGapCentreAxis].stStatus.bFwEnabled := TRUE;
END_IF

//GAP CENTRE BACKWARD LIMIT
IF GVL.astAxes[nIdPositiveAxis].stStatus.bBwEnabled = FALSE OR GVL.astAxes[nIdNegativeAxis].stStatus.bBwEnabled = FALSE THEN
    //GVL.astAxes[nIdGapCentreAxis].stInputs.bLimitBwd := FALSE;
    GVL.astAxes[nIdGapCentreAxis].stStatus.bBwEnabled := FALSE;
ELSE
    //GVL.astAxes[nIdGapCentreAxis].stInputs.bLimitBwd := TRUE;
    GVL.astAxes[nIdGapCentreAxis].stStatus.bBwEnabled := TRUE;
END_IF
END_ACTION

ACTION actVirtualAxisPositions:

(*Calculate virtual axis positions and convert to UDINT.
Conversion to UDINT is prohibited if it would exceed UDINT max value of 4,294,967,295.
If this is not done, it can cause overflow when connected to the encoder input and hard-crash the PLC which will only recover with a power cycle.
To preserve decimal position data of the LREAL (i.e. anything <1mm) it is necessary to scale the value before converting to UDINT.
This can be reversed with the correct scaling at the NC encoder level.
*)
fGapSize := GVL.astAxes[nIdPositiveAxis].stStatus.fActPosition - GVL.astAxes[nIdNegativeAxis].stStatus.fActPosition;
fGapCentre := (GVL.astAxes[nIdPositiveAxis].stStatus.fActPosition + GVL.astAxes[nIdNegativeAxis].stStatus.fActPosition)/2;


    IF ABS(fGapSize) < 100000 THEN
        nGapSizeEncoder := LREAL_TO_UDINT(fGapSize*fEncoderScaling);
    END_IF
    IF ABS(fGapCentre) < 100000 THEN
        nGapCentreEncoder := LREAL_TO_UDINT(fGapCentre*fEncoderScaling);
    END_IF
END_ACTION

ACTION Setpoint_AllDisabled:
fPosSetpointPositiveAxis := fPosSetpointPositiveAxis;
fPosSetpointNegativeAxis := fPosSetpointNegativeAxis;            
fVeloSetpointPositiveAxis := 0;
fVeloSetpointNegativeAxis := 0;

fbSetpointGenEnableGapCentreAxis.Execute:= TRUE;
fbSetpointGenEnableGapCentreAxis(Axis:= GVL.astAxes[nIdGapCentreAxis].Axis);
fPosSetpointGapCentreAxis := (GVL.astAxes[nIdPositiveAxis].Axis.NcToPlc.ActPos + GVL.astAxes[nIdNegativeAxis].Axis.NcToPlc.ActPos)/2;
fVeloSetpointGapCentreAxis := fVeloSetpointGapCentreAxis_New;


actHaltAllAxes();
END_ACTION

ACTION Setpoint_NegativeDisabled:
fPosSetpointPositiveAxis := GVL.astAxes[nIdGapSizeAxis].Axis.NcToPlc.SetPos + GVL.astAxes[nIdNegativeAxis].Axis.NcToPlc.ActPos;
fPosSetpointNegativeAxis := fPosSetpointNegativeAxis;
fVeloSetpointPositiveAxis := GVL.astAxes[nIdGapSizeAxis].Axis.NcToPlc.SetVelo;
fVeloSetpointNegativeAxis := 0;
            
fbSetpointGenEnableGapCentreAxis.Execute:= TRUE;
fbSetpointGenEnableGapCentreAxis(Axis:= GVL.astAxes[nIdGapCentreAxis].Axis);
fPosSetpointGapCentreAxis := fGapCentre;
fVeloSetpointGapCentreAxis := fVeloSetpointGapCentreAxis_New;
END_ACTION

ACTION Setpoint_Normal:
fPosSetpointPositiveAxis := fPosSetpointPositiveAxis_Nominal;
fPosSetpointNegativeAxis := fPosSetpointNegativeAxis_Nominal;
fVeloSetpointPositiveAxis := fVeloSetpointPositiveAxis_New;
fVeloSetpointNegativeAxis := fVeloSetpointNegativeAxis_New;
END_ACTION

ACTION Setpoint_PositiveDisabled:
fPosSetpointPositiveAxis := fPosSetpointPositiveAxis;
fPosSetpointNegativeAxis := GVL.astAxes[nIdPositiveAxis].Axis.NcToPlc.ActPos - GVL.astAxes[nIdGapSizeAxis].Axis.NcToPlc.SetPos;
fVeloSetpointPositiveAxis := 0;
fVeloSetpointNegativeAxis := GVL.astAxes[nIdGapSizeAxis].Axis.NcToPlc.SetVelo;
            
fbSetpointGenEnableGapCentreAxis.Execute:= TRUE;
fbSetpointGenEnableGapCentreAxis(Axis:= GVL.astAxes[nIdGapCentreAxis].Axis);
fPosSetpointGapCentreAxis := fGapCentre;
fVeloSetpointGapCentreAxis := fVeloSetpointGapCentreAxis_New;
END_ACTION

END_FUNCTION_BLOCK

(* stored: Version 1.1.0.1, ProductVersion 3.1.4024.11
   POU FB_SlitPairV2: Id {ff4013b1-472a-4f42-a6c8-2711712ac06d}, SpecialFunc None
   Folder Setpoint_Generator_Actions: Id {8e494922-e7c2-4daa-80b3-ea89aa78df74}
   Action actCalculateSetpointDirections: Id {7783e346-7fab-40d5-bab7-fe46a8c2f785}
   Action actCalculateSetpointPositions: Id {08e35b97-914a-4ccc-a3af-6b7cd8e60439}
   Action actCalculateSetpointVelocities: Id {59813eea-6905-4661-a8f3-10b16a472979}
   Action actGeneratorEnableDisable: Id {d59f6d39-50eb-4cb0-8d9d-b62df150c5a5}
   Action actHaltAllAxes: Id {f2afb93d-4a80-499a-b8ec-4e673220e7ad}
   Action actLimitState: Id {76476edf-1ca7-4d8b-8b71-a3d45cf78601}
   Action actVirtualAxisEnable: Id {d8729d12-361d-472b-8974-5b566dad7d06}
   Action actVirtualAxisLimits: Id {436d835a-8846-47e9-922d-a1df63469a25}
   Action actVirtualAxisPositions: Id {4ef557a2-3171-4a03-98ba-14f2cd3ef5ec}
   Action Setpoint_AllDisabled: Id {8d0131b7-d925-4748-8e58-1076d969b851}
   Action Setpoint_NegativeDisabled: Id {9ce73458-d767-47d6-a68a-e8346e22f1ca}
   Action Setpoint_Normal: Id {2ee67b84-83cd-44fc-84d0-218d8dc38cfa}
   Action Setpoint_PositiveDisabled: Id {1b4e9e96-8a89-4887-bc05-9c26a4b38f02} *)
